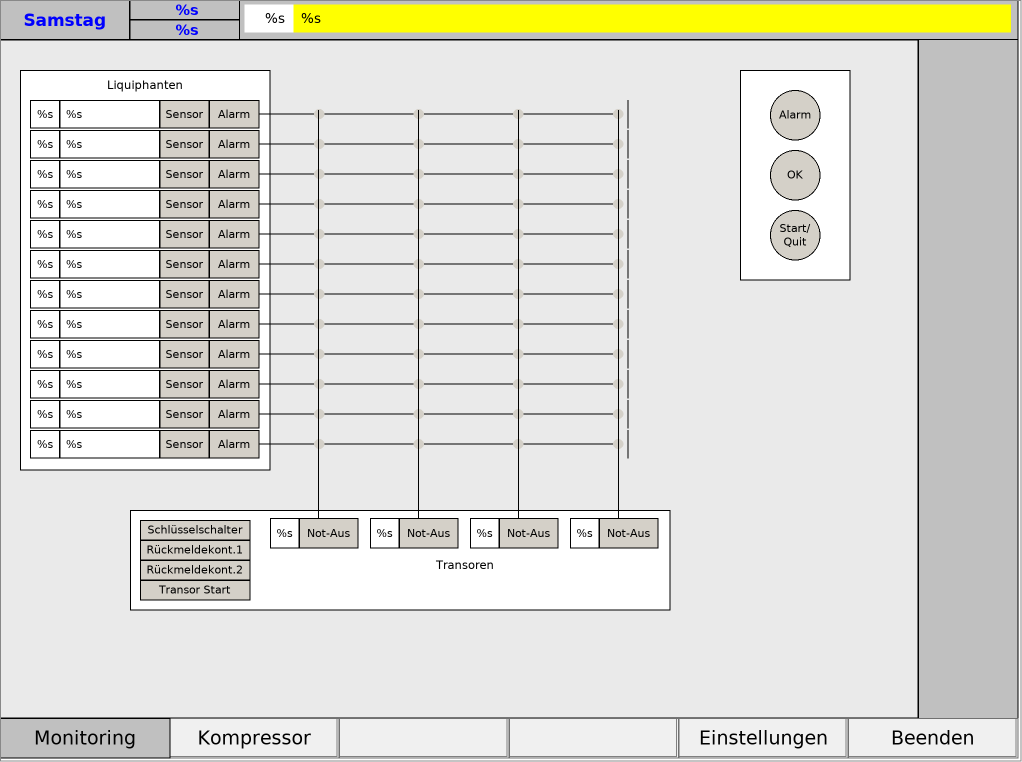
VISUALIZATION V_Monitoring  // 1022x762
    Frame (0,0 1020x760)
        shows V_Main_PC()
    Rectangle (20,70 250x400)
    Rectangle (130,510 540x100)
    Rectangle (0,718 170x40), "Monitoring"
    Frame (30,100 600x30)
        shows V_LiquidSensorState(IOfbLiquidSensor := PLC_PRG.fbLiquidMonitoring.fbLiquidSensor[1])
    Frame (30,130 600x30)
        shows V_LiquidSensorState(IOfbLiquidSensor := PLC_PRG.fbLiquidMonitoring.fbLiquidSensor[2])
    Frame (30,160 600x30)
        shows V_LiquidSensorState(IOfbLiquidSensor := PLC_PRG.fbLiquidMonitoring.fbLiquidSensor[3])
    Frame (30,190 600x30)
        shows V_LiquidSensorState(IOfbLiquidSensor := PLC_PRG.fbLiquidMonitoring.fbLiquidSensor[4])
    Frame (30,220 600x30)
        shows V_LiquidSensorState(IOfbLiquidSensor := PLC_PRG.fbLiquidMonitoring.fbLiquidSensor[5])
    Frame (30,250 600x30)
        shows V_LiquidSensorState(IOfbLiquidSensor := PLC_PRG.fbLiquidMonitoring.fbLiquidSensor[6])
    Frame (30,280 600x30)
        shows V_LiquidSensorState(IOfbLiquidSensor := PLC_PRG.fbLiquidMonitoring.fbLiquidSensor[7])
    Frame (30,310 600x30)
        shows V_LiquidSensorState(IOfbLiquidSensor := PLC_PRG.fbLiquidMonitoring.fbLiquidSensor[8])
    Frame (30,340 600x30)
        shows V_LiquidSensorState(IOfbLiquidSensor := PLC_PRG.fbLiquidMonitoring.fbLiquidSensor[9])
    Frame (30,370 600x30)
        shows V_LiquidSensorState(IOfbLiquidSensor := PLC_PRG.fbLiquidMonitoring.fbLiquidSensor[10])
    Frame (30,400 600x30)
        shows V_LiquidSensorState(IOfbLiquidSensor := PLC_PRG.fbLiquidMonitoring.fbLiquidSensor[11])
    Frame (30,430 600x30)
        shows V_LiquidSensorState(IOfbLiquidSensor := PLC_PRG.fbLiquidMonitoring.fbLiquidSensor[12])
    Frame (270,110 90x440)
        shows V_LiquidTransorState(IOfbTransor := PLC_PRG.fbLiquidMonitoring.fbTransor[1])
    Frame (370,110 90x440)
        shows V_LiquidTransorState(IOfbTransor := PLC_PRG.fbLiquidMonitoring.fbTransor[2])
    Frame (470,110 90x440)
        shows V_LiquidTransorState(IOfbTransor := PLC_PRG.fbLiquidMonitoring.fbTransor[3])
    Frame (570,110 90x440)
        shows V_LiquidTransorState(IOfbTransor := PLC_PRG.fbLiquidMonitoring.fbTransor[4])
    Rectangle (270,550 390x30), "Transoren"
    Rectangle (30,70 230x30), "Liquiphanten"
    Rectangle (740,70 110x210)
    Ellipse (770,90 50x50), "Alarm", colour toggle: PLC_PRG.fbLiquidMonitoring.QbLMStatusAlarm
    Ellipse (770,150 50x50), "OK", colour toggle: PLC_PRG.fbLiquidMonitoring.QbLMStatusOK
    Ellipse (770,210 50x50), "Start/ Quit", tooltip "Alarm quittieren und Transoren starten", colour toggle: PLC_PRG.fbLiquidMonitoring.QbLMStartQuit
        tap PLC_PRG.fbLiquidMonitoring.VbStartQuit
    Rectangle (140,520 110x20), "Schlüsselschalter", colour toggle: PLC_PRG.fbLiquidMonitoring.IbKeySwitch
    Rectangle (140,540 110x20), "Rückmeldekont.1", colour toggle: PLC_PRG.fbLiquidMonitoring.IbContactorResponse1
    Rectangle (140,560 110x20), "Rückmeldekont.2", colour toggle: PLC_PRG.fbLiquidMonitoring.IbContactorResponse2
    Rectangle (140,580 110x20), "Transor Start", colour toggle: PLC_PRG.fbLiquidMonitoring.QbStartTransor
END_VISUALIZATION

// ---- Visualizations/V_Logger.TcVIS
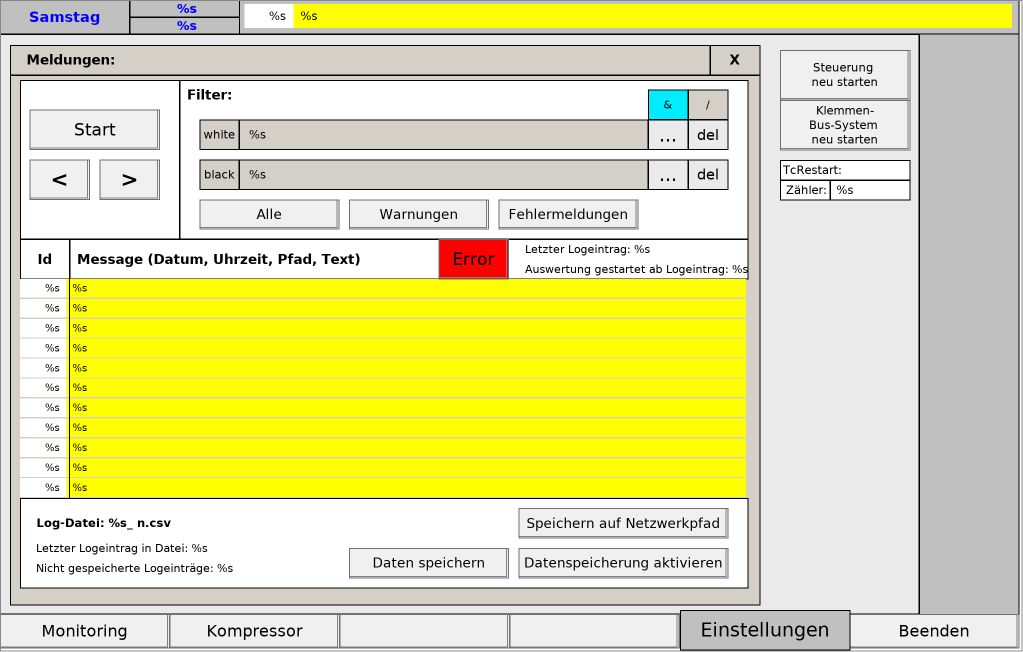
VISUALIZATION V_Logger  // 1023x652
    Frame (0,0 1021x650)
        shows V_Main_PC()
    Rectangle (680,610 170x40), "Einstellungen"
    Button (780,50 130x50), "Steuerung neu starten", invisible if: gfbSystemCX.tonStartUp.Q = 0
        OnMouseUp: change screen: V_TCReset
    Button (780,100 130x50), "Klemmen- Bus-System neu starten", invisible if: gfbSystemCX.tonStartUp.Q = 0
        OnMouseUp: change screen: V_ECReset
    Rectangle (10,75 750x530)
    Rectangle (10,45 700x30), "Meldungen:"
    Rectangle (710,45 50x30), "X"
        OnMouseClick: change screen: Previous 
    Rectangle (830,180 80x20), "%s", text variable: gfbSystemCX.nviTcRestartCnt
    Rectangle (780,160 130x20), "TcRestart:"
    Rectangle (780,180 50x20), "Zähler:"
    Frame (20,80 730x510)
        shows V_LoggerModul(fbLogger := gfbLogger)
END_VISUALIZATION

// ---- Visualizations/V_KomprWRG.TcVIS
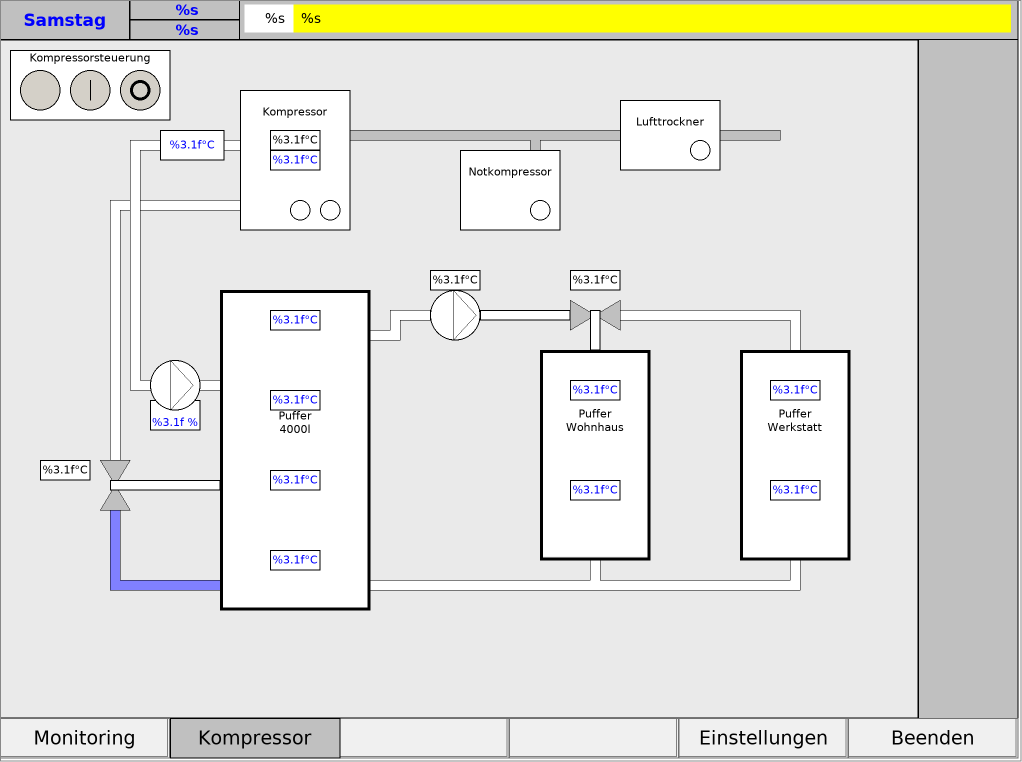
VISUALIZATION V_KomprWRG  // 1022x762
    Frame (0,0 1020x760)
        shows V_Main_PC()
    Polygon (330,130) (780,130) (780,140) (540,140) (540,150) (530,150) (530,140) (330,140)
    Polygon (570,300) (620,330) (620,300) (570,330) (570,320), colour toggle: PLC_PRG.fbKompressorSteuerung.QbVentilUmschWerkstatt
    Ellipse (430,290 50x50), colour toggle: PLC_PRG.fbKompressorSteuerung.QbUmwaelzpumpeWohnhaus
    Polygon (453,290) (476,315) (453,340) (453,327)
    Rectangle (480,310 90x10), colour toggle: PLC_PRG.fbKompressorSteuerung.QbUmwaelzpumpeWohnhaus
    Rectangle (590,310 10x40), colour toggle: PLC_PRG.fbKompressorSteuerung.QbVentilUmschWerkstatt
    Polygon (620,310) (800,310) (800,350) (790,350) (790,320) (620,320), colour toggle: PLC_PRG.fbKompressorSteuerung.QbUmwaelzpumpeWohnhaus and not PLC_PRG.fbKompressorSteuerung.QbVentilUmschWerkstatt
    Polygon (370,580) (390,580) (410,580) (590,580) (590,560) (600,560) (600,580) (790,580) (790,560) (800,560) (800,580) (800,590) (400,590) (390,590) (370,590), colour toggle: PLC_PRG.fbKompressorSteuerung.QbUmwaelzpumpeWohnhaus
    Rectangle (150,400 50x30), "%3.1f %", text variable: PLC_PRG.fbKompressorSteuerung.fbAnalogOutUmwaelzpumpeWRG.INrValue * 100
    Rectangle (240,90 110x140), "Kompressor"
    Rectangle (460,150 100x80), "Notkompressor"
    Rectangle (620,100 100x70), "Lufttrockner"
    Ellipse (690,140 20x20), colour toggle: PLC_PRG.fbKompressorSteuerung.QbLufttrockner
    Ellipse (530,200 20x20), colour toggle: PLC_PRG.fbKompressorSteuerung.QbNotKompressor
    Ellipse (320,200 20x20), colour toggle: PLC_PRG.fbKompressorSteuerung.QbKompressor
    Ellipse (290,200 20x20), tooltip "Störung", colour toggle: PLC_PRG.fbKompressorSteuerung.IbStoerung
    Polygon (100,510) (130,460) (100,460) (130,510) (130,510), colour toggle: PLC_PRG.fbKompressorSteuerung.QbVentilSchnellauflWRG
    Rectangle (110,480 110x10), colour toggle: PLC_PRG.fbKompressorSteuerung.QbVentilSchnellauflWRG
    Polygon (110,510) (110,590) (220,590) (220,580) (120,580) (120,510), colour toggle: PLC_PRG.fbKompressorSteuerung.QbVentilSchnellauflWRG
    Polygon (240,210) (120,210) (120,460) (110,460) (110,200) (240,200), colour toggle: PLC_PRG.fbKompressorSteuerung.QbUmwaelzpumpeWRG
    Polygon (240,140) (130,140) (130,390) (220,390) (220,380) (140,380) (140,150) (240,150), colour toggle: PLC_PRG.fbKompressorSteuerung.QbUmwaelzpumpeWRG
    Ellipse (150,360 50x50), colour toggle: PLC_PRG.fbKompressorSteuerung.QbUmwaelzpumpeWRG
    Polygon (170,360) (193,385) (170,410) (170,397)
    Rectangle (160,130 64x30), "%3.1f°C", text variable: gfbTemp31_KomprWRG_Ruecklauf.OUTrValue
    Rectangle (270,150 50x20), "%3.1f°C", text variable: gfbTemp32_KomprWRG_Vorlauf.OUTrValue
    Rectangle (40,460 50x20), "%3.1f°C", tooltip "Temperatur, Umschaltung Schnellaufladung", text variable: PLC_PRG.fbKompressorSteuerung.VrKomprWRG_TempSchnellaufl
        OnMouseClick: write the text variable via Default, min 20, max 70
    Rectangle (270,130 50x20), "%3.1f°C", tooltip "Solltemperatur Vorlauf", text variable: PLC_PRG.fbKompressorSteuerung.VrKomprWRG_TempVorlaufSollwert
        OnMouseClick: write the text variable via Default, min 20, max 80
    Rectangle (430,270 50x20), "%3.1f°C", tooltip "Temperatur, Umschaltung zum Wohnhaus", text variable: PLC_PRG.fbKompressorSteuerung.VrKomprWRG_TempUmschaltZurWohnh
        OnMouseClick: write the text variable via Default, min 20, max 70
    Rectangle (570,270 50x20), "%3.1f°C", tooltip "Temperatur, Umschaltung zur Werkstatt", text variable: PLC_PRG.fbKompressorSteuerung.VrKomprWRG_TempUmschaltZurWerkst
        OnMouseClick: write the text variable via Default, min 20, max 70
    Polygon (430,310) (430,320) (400,320) (400,340) (370,340) (370,330) (390,330) (390,310), colour toggle: PLC_PRG.fbKompressorSteuerung.QbUmwaelzpumpeWohnhaus
    Rectangle (10,50 160x70), "Kompressorsteuerung"
    Ellipse (20,70 40x40), tooltip "Störung", colour toggle: PLC_PRG.fbKompressorSteuerung.QbLMStatus
    Ellipse (70,70 40x40), tooltip "Störung", colour toggle: PLC_PRG.fbKompressorSteuerung.VbStart
        tap PLC_PRG.fbKompressorSteuerung.VbStart
    Ellipse (120,70 40x40), tooltip "Störung", colour toggle: PLC_PRG.fbKompressorSteuerung.VbStop
        tap PLC_PRG.fbKompressorSteuerung.VbStop
    RoundedRectangle (222,520 146x88), colour variable: gfbTemp14_Puffer4000_unten.VdiColourOfTemperature
    Ellipse (130,80 20x20)
    Line (90,80) (90,100)
    RoundedRectangle (222,440 146x95), colour variable: gfbTemp13_Puffer4000_mitte.VdiColourOfTemperature
    RoundedRectangle (222,360 146x95), colour variable: gfbTemp12_Puffer4000_oben.VdiColourOfTemperature
    RoundedRectangle (222,292 146x85), colour variable: gfbTemp11_Puffer4000_Brauchw.VdiColourOfTemperature
    RoundedRectangle (220,290 150x320), "Puffer 4000l"
    Rectangle (270,390 50x20), "%3.1f°C", text variable: gfbTemp12_Puffer4000_oben.OUTrValue
    Rectangle (270,470 50x20), "%3.1f°C", text variable: gfbTemp13_Puffer4000_mitte.OUTrValue
    Rectangle (270,550 50x20), "%3.1f°C", text variable: gfbTemp14_Puffer4000_unten.OUTrValue
    Rectangle (270,310 50x20), "%3.1f°C", text variable: gfbTemp11_Puffer4000_Brauchw.OUTrValue
    RoundedRectangle (742,450 106x108), colour variable: gfbTemp24_PufferWerkst_unten.VdiColourOfTemperature
    RoundedRectangle (742,352 106x110), colour variable: gfbTemp23_PufferWerkst_oben.VdiColourOfTemperature
    RoundedRectangle (740,350 110x210), "Puffer Werkstatt"
    Rectangle (770,480 50x20), "%3.1f°C", text variable: gfbTemp24_PufferWerkst_unten.OUTrValue
    Rectangle (770,380 50x20), "%3.1f°C", text variable: gfbTemp23_PufferWerkst_oben.OUTrValue
    RoundedRectangle (542,448 106x108), colour variable: gfbTemp22_PufferWohnh_unten.VdiColourOfTemperature
    RoundedRectangle (542,352 106x110), colour variable: gfbTemp21_PufferWohnh_oben.VdiColourOfTemperature
    Rectangle (570,480 50x20), "%3.1f°C", text variable: gfbTemp22_PufferWohnh_unten.OUTrValue
    Rectangle (570,380 50x20), "%3.1f°C", text variable: gfbTemp21_PufferWohnh_oben.OUTrValue
    RoundedRectangle (540,350 110x210), "Puffer Wohnhaus"
    Rectangle (170,718 170x40), "Kompressor"
END_VISUALIZATION

// ---- Visualizations/V_Einstellungen.TcVIS
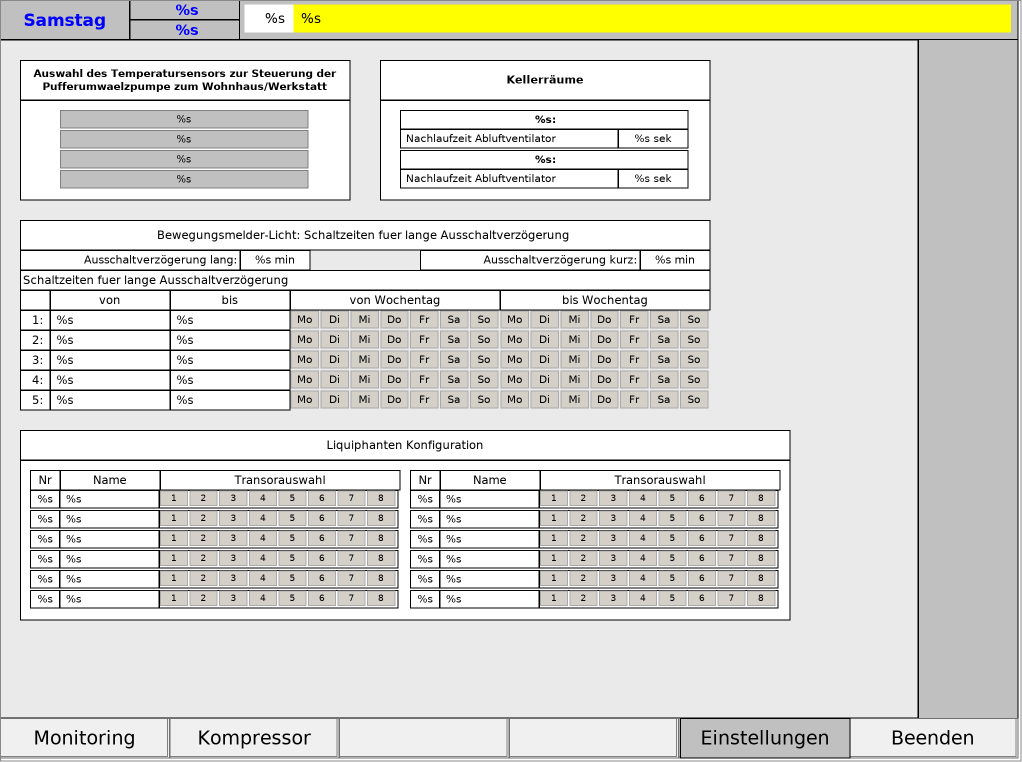
VISUALIZATION V_Einstellungen  // 1022x762
    Frame (0,0 1020x760)
        shows V_Main_PC()
    Rectangle (20,460 770x160)
    Rectangle (380,60 330x40), "Kellerräume", tooltip "Nach Abschalten des Bewegungsmelders läuft der Abluftventilator die hier eingestellte Zeit nach"
    Rectangle (380,100 330x100), tooltip "Nach Abschalten des Bewegungsmelders läuft der Abluftventilator die hier eingestellte Zeit nach"
    Rectangle (20,100 330x100), tooltip "Nach Abschalten des Bewegungsmelders läuft der Abluftventilator die hier eingestellte Zeit nach"
    Rectangle (20,60 330x40), "Auswahl des Temperatursensors zur Steuerung der Pufferumwaelzpumpe zum Wohnhaus/Werkstatt", tooltip "Nach Abschalten des Bewegungsmelders läuft der Abluftventilator die hier eingestellte Zeit nach"
    Frame (60,110 250x20)
        shows V_RadioButton(IN_Title := '4000l-Puffer Brauchw.', IN_iValue := 4, IO_iVar := PLC_PRG.fbKompressorSteuerung.ViWRGTempSensorSelect)
    Frame (60,130 250x20)
        shows V_RadioButton(IN_Title := '4000l-Puffer oben', IN_iValue := 3, IO_iVar := PLC_PRG.fbKompressorSteuerung.ViWRGTempSensorSelect)
    Frame (60,150 250x20)
        shows V_RadioButton(IN_Title := '4000l-Puffer mitte', IN_iValue := 2, IO_iVar := PLC_PRG.fbKompressorSteuerung.ViWRGTempSensorSelect)
    Frame (60,170 250x20)
        shows V_RadioButton(IN_Title := '4000l-Puffer unten', IN_iValue := 1, IO_iVar := PLC_PRG.fbKompressorSteuerung.ViWRGTempSensorSelect)
    Rectangle (50,290 120x20), "von"
    Rectangle (50,310 120x20), "%s", text variable: VnvstSwitchTimesLichtBWMtofLang.todHeizEin[1]
        OnMouseDown: write the text variable via Edit
    Rectangle (20,310 30x20), "1:"
    Rectangle (20,220 690x30), "Bewegungsmelder-Licht: Schaltzeiten fuer lange Ausschaltverzögerung"
    Rectangle (20,330 30x20), "2:"
    Rectangle (20,350 30x20), "3:"
    Rectangle (20,370 30x20), "4:"
    Rectangle (20,390 30x20), "5:"
    Rectangle (170,290 120x20), "bis"
    Rectangle (20,290 30x20)
    Rectangle (170,310 120x20), "%s", text variable: VnvstSwitchTimesLichtBWMtofLang.todHeizAus[1]
        OnMouseDown: write the text variable via Edit
    Rectangle (290,290 210x20), "von Wochentag"
    Rectangle (500,290 210x20), "bis Wochentag"
    Rectangle (50,330 120x20), "%s", text variable: VnvstSwitchTimesLichtBWMtofLang.todHeizEin[2]
        OnMouseDown: write the text variable via Edit
    Rectangle (170,330 120x20), "%s", text variable: VnvstSwitchTimesLichtBWMtofLang.todHeizAus[2]
        OnMouseDown: write the text variable via Edit
    Rectangle (50,350 120x20), "%s", text variable: VnvstSwitchTimesLichtBWMtofLang.todHeizEin[3]
        OnMouseDown: write the text variable via Edit
    Rectangle (170,350 120x20), "%s", text variable: VnvstSwitchTimesLichtBWMtofLang.todHeizAus[3]
        OnMouseDown: write the text variable via Edit
    Rectangle (50,370 120x20), "%s", text variable: VnvstSwitchTimesLichtBWMtofLang.todHeizEin[4]
        OnMouseDown: write the text variable via Edit
    Rectangle (170,370 120x20), "%s", text variable: VnvstSwitchTimesLichtBWMtofLang.todHeizAus[4]
        OnMouseDown: write the text variable via Edit
    Rectangle (50,390 120x20), "%s", text variable: VnvstSwitchTimesLichtBWMtofLang.todHeizEin[5]
        OnMouseDown: write the text variable via Edit
    Rectangle (170,390 120x20), "%s", text variable: VnvstSwitchTimesLichtBWMtofLang.todHeizAus[5]
        OnMouseDown: write the text variable via Edit
    Rectangle (20,270 690x20), "Schaltzeiten fuer lange Ausschaltverzögerung"
    Rectangle (240,250 70x20), "%s min", tooltip "Nach Abschalten des Bewegungsmelders läuft der Abluftventilator die hier eingestellte Zeit nach", text variable: VnvdiLichtTofLang
        OnMouseClick: write the text variable via Default, min 3, max 600
    Rectangle (20,250 220x20), "Ausschaltverzögerung lang:", tooltip "Nach Abschalten des Bewegungsmelders läuft der Abluftventilator die hier eingestellte Zeit nach"
    Rectangle (420,250 220x20), "Ausschaltverzögerung kurz:", tooltip "Nach Abschalten des Bewegungsmelders läuft der Abluftventilator die hier eingestellte Zeit nach"
    Rectangle (640,250 70x20), "%s min", tooltip "Nach Abschalten des Bewegungsmelders läuft der Abluftventilator die hier eingestellte Zeit nach", text variable: VnvdiLichtTofKurz
        OnMouseClick: write the text variable via Default, min 0, max 30
    Frame (290,390 210x20)
        shows V_WeekDay(eWeekDay := VnvstSwitchTimesLichtBWMtofLang.eDayOfWeekStart[5])
    Frame (500,390 210x20)
        shows V_WeekDay(eWeekDay := VnvstSwitchTimesLichtBWMtofLang.eDayOfWeekEnd[5])
    Frame (290,310 210x20)
        shows V_WeekDay(eWeekDay := VnvstSwitchTimesLichtBWMtofLang.eDayOfWeekStart[1])
    Frame (500,310 210x20)
        shows V_WeekDay(eWeekDay := VnvstSwitchTimesLichtBWMtofLang.eDayOfWeekEnd[1])
    Frame (290,330 210x20)
        shows V_WeekDay(eWeekDay := VnvstSwitchTimesLichtBWMtofLang.eDayOfWeekStart[2])
    Frame (500,330 210x20)
        shows V_WeekDay(eWeekDay := VnvstSwitchTimesLichtBWMtofLang.eDayOfWeekEnd[2])
    Frame (290,350 210x20)
        shows V_WeekDay(eWeekDay := VnvstSwitchTimesLichtBWMtofLang.eDayOfWeekStart[3])
    Frame (500,350 210x20)
        shows V_WeekDay(eWeekDay := VnvstSwitchTimesLichtBWMtofLang.eDayOfWeekEnd[3])
    Frame (290,370 210x20)
        shows V_WeekDay(eWeekDay := VnvstSwitchTimesLichtBWMtofLang.eDayOfWeekStart[4])
    Frame (500,370 210x20)
        shows V_WeekDay(eWeekDay := VnvstSwitchTimesLichtBWMtofLang.eDayOfWeekEnd[4])
    Rectangle (680,718 170x40), "Einstellungen"
    Frame (400,150 290x40)
        shows V_WCRaum(IN_Title := 'WC Herren', IO_fbWCRaum := PLC_PRG.fbWCHerren)
    Frame (400,110 290x40)
        shows V_WCRaum(IN_Title := 'WC Damen', IO_fbWCRaum := PLC_PRG.fbWCDamen)
    Rectangle (20,430 770x30), "Liquiphanten Konfiguration"
    Rectangle (30,470 30x20), "Nr"
    Rectangle (160,470 240x20), "Transorauswahl"
    Rectangle (60,470 100x20), "Name"
    Frame (30,490 370x20)
        shows V_LiquidSensorCfg(iNumOfCh := PLC_PRG.fbLiquidMonitoring.iNUM_OF_TRANSORS, IOfbLiquidSensor := PLC_PRG.fbLiquidMonitoring.fbLiquidSensor[1])
    Frame (30,510 370x20)
        shows V_LiquidSensorCfg(iNumOfCh := PLC_PRG.fbLiquidMonitoring.iNUM_OF_TRANSORS, IOfbLiquidSensor := PLC_PRG.fbLiquidMonitoring.fbLiquidSensor[2])
    Frame (30,530 370x20)
        shows V_LiquidSensorCfg(iNumOfCh := PLC_PRG.fbLiquidMonitoring.iNUM_OF_TRANSORS, IOfbLiquidSensor := PLC_PRG.fbLiquidMonitoring.fbLiquidSensor[3])
    Frame (30,550 370x20)
        shows V_LiquidSensorCfg(iNumOfCh := PLC_PRG.fbLiquidMonitoring.iNUM_OF_TRANSORS, IOfbLiquidSensor := PLC_PRG.fbLiquidMonitoring.fbLiquidSensor[4])
    Frame (30,570 370x20)
        shows V_LiquidSensorCfg(iNumOfCh := PLC_PRG.fbLiquidMonitoring.iNUM_OF_TRANSORS, IOfbLiquidSensor := PLC_PRG.fbLiquidMonitoring.fbLiquidSensor[5])
    Frame (30,590 370x20)
        shows V_LiquidSensorCfg(iNumOfCh := PLC_PRG.fbLiquidMonitoring.iNUM_OF_TRANSORS, IOfbLiquidSensor := PLC_PRG.fbLiquidMonitoring.fbLiquidSensor[6])
    Frame (410,490 370x20)
        shows V_LiquidSensorCfg(iNumOfCh := PLC_PRG.fbLiquidMonitoring.iNUM_OF_TRANSORS, IOfbLiquidSensor := PLC_PRG.fbLiquidMonitoring.fbLiquidSensor[7])
    Frame (410,510 370x20)
        shows V_LiquidSensorCfg(iNumOfCh := PLC_PRG.fbLiquidMonitoring.iNUM_OF_TRANSORS, IOfbLiquidSensor := PLC_PRG.fbLiquidMonitoring.fbLiquidSensor[8])
    Rectangle (410,470 30x20), "Nr"
    Rectangle (540,470 240x20), "Transorauswahl"
    Rectangle (440,470 100x20), "Name"
    Frame (410,530 370x20)
        shows V_LiquidSensorCfg(iNumOfCh := PLC_PRG.fbLiquidMonitoring.iNUM_OF_TRANSORS, IOfbLiquidSensor := PLC_PRG.fbLiquidMonitoring.fbLiquidSensor[9])
    Frame (410,550 370x20)
        shows V_LiquidSensorCfg(iNumOfCh := PLC_PRG.fbLiquidMonitoring.iNUM_OF_TRANSORS, IOfbLiquidSensor := PLC_PRG.fbLiquidMonitoring.fbLiquidSensor[10])
    Frame (410,570 370x20)
        shows V_LiquidSensorCfg(iNumOfCh := PLC_PRG.fbLiquidMonitoring.iNUM_OF_TRANSORS, IOfbLiquidSensor := PLC_PRG.fbLiquidMonitoring.fbLiquidSensor[11])
    Frame (410,590 370x20)
        shows V_LiquidSensorCfg(iNumOfCh := PLC_PRG.fbLiquidMonitoring.iNUM_OF_TRANSORS, IOfbLiquidSensor := PLC_PRG.fbLiquidMonitoring.fbLiquidSensor[12])
END_VISUALIZATION
